FUNCTION_BLOCK FB_OperatingMode
VAR_INPUT
	PermissionHardware	:	BOOL;	//Permission hardware ready for operation
	PermissionSoftware	:	BOOL;	//Permission from safety machine ready for start
	E_Stop	:	BOOL;	//Button E-Stop
	OperatingModeManual	:	BOOL;	//Operating Mode manual is selected
	OperatingModeAutomatic	:	BOOL;	//Operating Mode automatic is selected
END_VAR
VAR_OUTPUT
	LEDStart	:	BOOL;	//Indicator to show state automatic start
	LEDStop	:	BOOL;	//Indicator to show state automatic stop
	LEDHome	:	BOOL;	//Indicator to show state automatic home
	LEDReset	:	BOOL;	//Indicator to show state reset
	LEDQuit	:	BOOL;	//Indicator to show state quit
END_VAR
VAR_IN_OUT
	HMIInterface	:	HMIInterfaceOperatingMode;
END_VAR
VAR
	statRisingEdgeAutomaticActivated	:	BOOL;	//Rising edge, used when Automatic is activated
	statOperatingMode	:	OperatingMode;
	statResetMethod	:	BOOL;
	statQuitMethod	:	BOOL;
	
	statHMIInterface	:	HMIInterfaceOperatingMode;
	statRisingEdgeManuelButtonPressedMachine	:	R_TRIG;
	statRisingEdgeManuelButtonPressedHMI	:	R_TRIG;
	statRisingEdgeAutomaticButtonPressedMachine	:	R_TRIG;
	statRisingEdgeAutomaticButtonPressedHMI	:	R_TRIG;
	statRisingEdgeAutomaticStartButtonPressedHMI	:	R_TRIG;
	statRisingEdgeAutomaticStopButtonPressedHMI	:	R_TRIG;
	statRisingEdgeAutomaticHomeButtonPressedHMI	:	R_TRIG;
END_VAR

(*===================== HMI-Interface umladen =====================*)
statHMIInterface := HMIInterface;
(*===================== Betriebsartenwahl =====================*)
statRisingEdgeManuelButtonPressedMachine(CLK := OperatingModeManual);
statRisingEdgeManuelButtonPressedHMI(CLK := statHMIInterface.HMIToPLC.Manuel.IsSelected);
statRisingEdgeAutomaticButtonPressedMachine(CLK := OperatingModeAutomatic);
statRisingEdgeAutomaticButtonPressedHMI(CLK := statHMIInterface.HMIToPLC.Automatic.IsSelected);
(*===================== Operating Manual =====================*)
statHMIInterface.PLCToHMI.Manuel.PreconditionsFullfilled := TRUE;
IF statRisingEdgeManuelButtonPressedMachine.Q OR
	(statRisingEdgeManuelButtonPressedHMI.Q AND statHMIInterface.PLCToHMI.Manuel.PreconditionsFullfilled)
	THEN
	statOperatingMode.ManuelIsActive := TRUE;
	statOperatingMode.AutomaticIsActive := FALSE;
END_IF
// statOperatingMode.ManuelIsActive := OperatingModeManual; 
(*===================== Operating Automatic =====================*)
statHMIInterface.PLCToHMI.Automatic.PreconditionsFullfilled := TRUE;
// statOperatingMode.AutomaticIsActive := OperatingModeAutomatic;
IF statRisingEdgeAutomaticButtonPressedMachine.Q OR
	(statRisingEdgeAutomaticButtonPressedHMI.Q AND statHMIInterface.PLCToHMI.Manuel.PreconditionsFullfilled)
	THEN
	statOperatingMode.AutomaticIsActive := TRUE;
	statOperatingMode.ManuelIsActive := FALSE;
END_IF
(*===================== HMI-Interface Betriebsarten =====================*)
statHMIInterface.PLCToHMI.Automatic.IsActive := statOperatingMode.AutomaticIsActive; 
statHMIInterface.PLCToHMI.Manuel.IsActive := statOperatingMode.ManuelIsActive;
(*===================== E-Stop is active =====================*)
statOperatingMode.EStop.PreconditionsFullfilled := TRUE;
statOperatingMode.EStop.IsActive := NOT E_Stop AND statOperatingMode.EStop.PreconditionsFullfilled;
(*===================== Reset is active =====================*)
statOperatingMode.Reset.PreconditionsFullfilled := TRUE;
statHMIInterface.PLCToHMI.Reset.PreconditionsFullfilled := statOperatingMode.Reset.PreconditionsFullfilled;
statOperatingMode.Reset.IsActive := (statResetMethod OR
									 statHMIInterface.HMIToPLC.Reset.IsSelected) AND 
									statOperatingMode.Reset.PreconditionsFullfilled;
statHMIInterface.PLCToHMI.Reset.IsActive := statOperatingMode.Reset.IsActive; 
(*===================== Quit is active =====================*)
statOperatingMode.Quit.PreconditionsFullfilled := TRUE;
statHMIInterface.PLCToHMI.Quit.PreconditionsFullfilled := statOperatingMode.Quit.PreconditionsFullfilled; 
statOperatingMode.Quit.IsActive := (statQuitMethod OR
									statHMIInterface.HMIToPLC.Quit.IsSelected) AND 
									statOperatingMode.Quit.PreconditionsFullfilled;
statHMIInterface.PLCToHMI.Quit.IsActive := statOperatingMode.Quit.IsActive; 
(*===================== Automatic Start is active =====================*)
statRisingEdgeAutomaticStartButtonPressedHMI(CLK := statHMIInterface.HMIToPLC.AutomaticStart.IsSelected);
statOperatingMode.AutomaticStart.PreconditionsFullfilled := PermissionHardware AND PermissionSoftware AND
												  			E_Stop AND NOT statOperatingMode.Reset.IsActive AND NOT
												  			statOperatingMode.AutomaticHome.IsActive AND NOT
															statOperatingMode.Fault.IsActive AND
												  			statOperatingMode.AutomaticIsActive;
statHMIInterface.PLCToHMI.AutomaticStart.PreconditionsFullfilled := statOperatingMode.AutomaticStart.PreconditionsFullfilled;
statOperatingMode.AutomaticStart.IsActive := (statOperatingMode.AutomaticStart.IsActive OR
											  statRisingEdgeAutomaticStartButtonPressedHMI.Q) AND
											  statOperatingMode.AutomaticStart.PreconditionsFullfilled;
IF statOperatingMode.AutomaticStart.IsActive AND statRisingEdgeAutomaticStartButtonPressedHMI.Q THEN
	statOperatingMode.AutomaticStop.IsActive := FALSE;
END_IF
statHMIInterface.PLCToHMI.AutomaticStart.IsActive := statOperatingMode.AutomaticStart.IsActive;
(*===================== Automatic Stop is active =====================*)
statRisingEdgeAutomaticStopButtonPressedHMI(CLK := statHMIInterface.HMIToPLC.AutomaticStop.IsSelected);
statOperatingMode.AutomaticStop.PreconditionsFullfilled := NOT statOperatingMode.AutomaticHome.IsActive;
statHMIInterface.PLCToHMI.AutomaticStop.PreconditionsFullfilled := statOperatingMode.AutomaticStop.PreconditionsFullfilled;
statOperatingMode.AutomaticStop.IsActive := ((statOperatingMode.AutomaticStop.IsActive OR statRisingEdgeAutomaticStopButtonPressedHMI.Q) AND
											 statOperatingMode.AutomaticStop.PreconditionsFullfilled) OR
											 statOperatingMode.ManuelIsActive OR statOperatingMode.Fault.IsActive OR 
											 (statOperatingMode.AutomaticIsActive AND (NOT PermissionHardware OR NOT PermissionSoftware)) OR
											  statOperatingMode.EStop.IsActive OR statOperatingMode.Reset.IsActive;
statHMIInterface.PLCToHMI.AutomaticStop.IsActive := statOperatingMode.AutomaticStop.IsActive;
IF statOperatingMode.AutomaticIsActive AND NOT statRisingEdgeAutomaticActivated THEN
	statRisingEdgeAutomaticActivated := TRUE;
	statOperatingMode.AutomaticStop.IsActive := TRUE;
ELSIF statOperatingMode.ManuelIsActive AND statRisingEdgeAutomaticActivated THEN
	statRisingEdgeAutomaticActivated := FALSE;
END_IF
IF statOperatingMode.AutomaticStop.IsActive AND statRisingEdgeAutomaticStopButtonPressedHMI.Q THEN
	statOperatingMode.AutomaticStop.IsActive := TRUE;
	statOperatingMode.AutomaticStart.IsActive := FALSE;
	statOperatingMode.AutomaticHome.IsActive := FALSE;
END_IF
(*===================== Automatic Home is active =====================*)
statRisingEdgeAutomaticHomeButtonPressedHMI(CLK := statHMIInterface.HMIToPLC.AutomaticHome.IsSelected);
statOperatingMode.AutomaticHome.IsReached := statOperatingMode.AutomaticHome.AllMachinesInHome;
IF statOperatingMode.AutomaticHome.IsReached THEN
	StateOperatingMode.AutomaticStop.IsActive := TRUE;
END_IF
statOperatingMode.AutomaticHome.PreconditionsFullfilled := PermissionHardware AND PermissionSoftware AND
												  			E_Stop AND NOT statOperatingMode.Reset.IsActive AND
												  			statOperatingMode.AutomaticIsActive AND NOT
														   statOperatingMode.AutomaticHome.IsReached;
statHMIInterface.PLCToHMI.AutomaticHome.PreconditionsFullfilled := statOperatingMode.AutomaticHome.PreconditionsFullfilled; 
statOperatingMode.AutomaticHome.IsActive := (statOperatingMode.AutomaticHome.IsActive OR
											statRisingEdgeAutomaticHomeButtonPressedHMI.Q) AND
											statOperatingMode.AutomaticHome.PreconditionsFullfilled;
IF statOperatingMode.AutomaticHome.IsActive AND statRisingEdgeAutomaticHomeButtonPressedHMI.Q THEN
	statOperatingMode.AutomaticHome.IsActive := TRUE;
	statOperatingMode.AutomaticStart.IsActive := FALSE;
	statOperatingMode.AutomaticStop.IsActive := FALSE;
END_IF
statHMIInterface.PLCToHMI.AutomaticHome.IsActive := statOperatingMode.AutomaticHome.IsActive; 
(*===================== Outputs =====================*)
LEDStart := statOperatingMode.AutomaticStart.IsActive;
LEDStop := statOperatingMode.AutomaticStop.IsActive;	
LEDHome := statOperatingMode.AutomaticHome.IsActive;	
LEDReset := statOperatingMode.Reset.IsActive;
LEDQuit	:= statOperatingMode.Quit.IsActive;
HMIInterface := statHMIInterface;

METHOD Homeing_On
VAR_INPUT
	ButtonHome	:	BOOL;
END_VAR
IF ButtonHome AND statOperatingMode.AutomaticStart.PreconditionsFullfilled AND NOT 
statOperatingMode.AutomaticHome.IsReached
THEN
	statOperatingMode.AutomaticStart.IsActive := FALSE;
	statOperatingMode.AutomaticStop.IsActive := FALSE;
	statOperatingMode.AutomaticHome.IsActive := TRUE;
END_IF
END_METHOD

METHOD PUBLIC Quit_On
VAR_INPUT
	ButtonQuit	:	BOOL;
END_VAR
IF ButtonQuit THEN
	statQuitMethod := TRUE;
ELSE
	statQuitMethod := FALSE;
END_IF
END_METHOD

METHOD PUBLIC Reset_on
VAR_INPUT
	ButtonReset	:	BOOL;
END_VAR
IF ButtonReset THEN
	statResetMethod := TRUE;
ELSE
	statResetMethod := FALSE;
END_IF
END_METHOD

METHOD PUBLIC Start_On
VAR_INPUT
	ButtonStart	:	BOOL;
END_VAR
IF ButtonStart AND statOperatingMode.AutomaticStart.PreconditionsFullfilled THEN
	statOperatingMode.AutomaticStart.IsActive := TRUE;
	statOperatingMode.AutomaticStop.IsActive := FALSE;
END_IF
END_METHOD

PROPERTY PUBLIC StateOperatingMode : REFERENCE TO OperatingMode
GET
StateOperatingMode REF= statOperatingMode;
END_GET
SET
statOperatingMode := StateOperatingMode;
END_SET
END_PROPERTY

METHOD PUBLIC Stop_On
VAR_INPUT
	ButtonStop	:	BOOL;
END_VAR
IF NOT ButtonStop AND statOperatingMode.AutomaticStart.PreconditionsFullfilled THEN
	statOperatingMode.AutomaticStart.IsActive := FALSE;
	statOperatingMode.AutomaticStop.IsActive := TRUE;
	statOperatingMode.AutomaticHome.IsActive := FALSE;
END_IF
END_METHOD

END_FUNCTION_BLOCK

(* stored: Version 1.1.0.1
   POU FB_OperatingMode: Id {c3dad087-efd8-4126-a802-e979de0f57d4}, SpecialFunc None
   Method Homeing_On: Id {7e62c1e5-310d-4727-8e63-27ba151a87a7}
   Method Quit_On: Id {7bf0d568-ee8b-41a5-90b0-b7945116ee25}
   Method Reset_on: Id {d2d797fd-82b1-4966-a207-58b034b34877}
   Method Start_On: Id {3354be3e-6726-4d80-9078-ae6449d88d6f}
   Property StateOperatingMode: Id {1c9be228-6bb8-46d1-a5b1-916f8552ece2}
   Get Get: Id {d0141e4b-206b-4b51-8a7a-654fc4ae35ce}
   Set Set: Id {c9478dc0-de45-4077-b675-ff8f777460cd}
   Method Stop_On: Id {916474fd-677f-4f1e-b324-eebd14fbfbbc} *)
